// TIA Portal V19 export
DATA_BLOCK "_IOL_VMrd_PointerInfo"   // DB23
TITLE = Info to construct pointer to Valve Monitoring Read parameters
{ S7_Optimized_Access := 'TRUE' }
// stored: AutoNumber false, MemoryReserve 0
   VAR RETAIN
      ACT : "_IOL_VMrdParInterface";
      acInt : Array[0..31] of "_IOL_VMrdParInterface";   // Process Object pointers
   END_VAR
BEGIN
   ACT.dataStore.dbno := 500;
   acInt[3..4].ia.dbno := 501;
   acInt[5..7].ia.dbno := 502;
   acInt[8..12].ia.dbno := 503;
   acInt[17..18].ia.dbno := 504;
   acInt[19].ia.dbno := 502;
   acInt[20..22].ia.dbno := 504;
   acInt[25].ia.dbno := 504;
   acInt[3..4].ia.al := 124;
   acInt[5..7].ia.al := 144;
   acInt[8..12].ia.al := 124;
   acInt[17..18].ia.al := 124;
   acInt[19].ia.al := 144;
   acInt[20..22].ia.al := 124;
   acInt[25].ia.al := 124;
   acInt[0].dataStore.dbno := 500;
   acInt[3..12].dataStore.dbno := 500;
   acInt[17..22].dataStore.dbno := 500;
   acInt[25].dataStore.dbno := 500;
   acInt[4].dataStore.sta := 40;
   acInt[5].dataStore.sta := 80;
   acInt[6].dataStore.sta := 120;
   acInt[7].dataStore.sta := 160;
   acInt[8].dataStore.sta := 200;
   acInt[9].dataStore.sta := 240;
   acInt[10].dataStore.sta := 280;
   acInt[11].dataStore.sta := 320;
   acInt[12].dataStore.sta := 360;
   acInt[17].dataStore.sta := 440;
   acInt[18].dataStore.sta := 480;
   acInt[19].dataStore.sta := 520;
   acInt[20].dataStore.sta := 560;
   acInt[21].dataStore.sta := 600;
   acInt[22].dataStore.sta := 640;
   acInt[25].dataStore.sta := 40;
   acInt[3..12].dataStore.al := 40;
   acInt[17..22].dataStore.al := 40;
   acInt[25].dataStore.al := 680;
END_DATA_BLOCK
